{attribute addProperty BoxType "KL6401-0002"}
{attribute addProperty Id "Parameter_StatusAT %I*UINT000Parameter_Input_Data_1AT %I*UDINT000Parameter_Input_Data_2AT %I*UDINT000Parameter_Input_Data_3AT %I*UDINT000Parameter_Input_Data_4AT %I*UDINT000Parameter_Input_Data_5AT %I*UDINT000Parameter_Input_Data_6AT %I*UDINT000Parameter_Input_Data_7AT %I*UDINT000Parameter_Input_Data_8AT %I*UDINT000Parameter_TypeAT %I*USINT000LON_StatusAT %I*USINT000Parameter_ControlAT %Q*UINT000Parameter_Output_Data_1AT %Q*UDINT000Parameter_Output_Data_2AT %Q*UDINT000Parameter_Output_Data_3AT %Q*UDINT000Parameter_Output_Data_4AT %Q*UDINT000Parameter_Output_Data_5AT %Q*UDINT000Parameter_Output_Data_6AT %Q*UDINT000Parameter_Output_Data_7AT %Q*UDINT000Parameter_Output_Data_8AT %Q*UDINT000CMDAT %Q*USINT000IdxAT %Q*USINT000"}
{attribute addProperty CRC "388522448"}
{attribute addProperty SizeInBites "0"}
{attribute addProperty SizeInBytes "0"}
TYPE Channel_172861D0 :
STRUCT
	{attribute addProperty Name "Parameter_Status"}
	Parameter_Status AT %I* : UINT;
	{attribute addProperty Name "Parameter_Input_Data_1"}
	Parameter_Input_Data_1 AT %I* : UDINT;
	{attribute addProperty Name "Parameter_Input_Data_2"}
	Parameter_Input_Data_2 AT %I* : UDINT;
	{attribute addProperty Name "Parameter_Input_Data_3"}
	Parameter_Input_Data_3 AT %I* : UDINT;
	{attribute addProperty Name "Parameter_Input_Data_4"}
	Parameter_Input_Data_4 AT %I* : UDINT;
	{attribute addProperty Name "Parameter_Input_Data_5"}
	Parameter_Input_Data_5 AT %I* : UDINT;
	{attribute addProperty Name "Parameter_Input_Data_6"}
	Parameter_Input_Data_6 AT %I* : UDINT;
	{attribute addProperty Name "Parameter_Input_Data_7"}
	Parameter_Input_Data_7 AT %I* : UDINT;
	{attribute addProperty Name "Parameter_Input_Data_8"}
	Parameter_Input_Data_8 AT %I* : UDINT;
	{attribute addProperty Name "Parameter_Type"}
	Parameter_Type AT %I* : USINT;
	{attribute addProperty Name "LON_Status"}
	LON_Status AT %I* : USINT;
	{attribute addProperty Name "Parameter_Control"}
	Parameter_Control AT %Q* : UINT;
	{attribute addProperty Name "Parameter_Output_Data_1"}
	Parameter_Output_Data_1 AT %Q* : UDINT;
	{attribute addProperty Name "Parameter_Output_Data_2"}
	Parameter_Output_Data_2 AT %Q* : UDINT;
	{attribute addProperty Name "Parameter_Output_Data_3"}
	Parameter_Output_Data_3 AT %Q* : UDINT;
	{attribute addProperty Name "Parameter_Output_Data_4"}
	Parameter_Output_Data_4 AT %Q* : UDINT;
	{attribute addProperty Name "Parameter_Output_Data_5"}
	Parameter_Output_Data_5 AT %Q* : UDINT;
	{attribute addProperty Name "Parameter_Output_Data_6"}
	Parameter_Output_Data_6 AT %Q* : UDINT;
	{attribute addProperty Name "Parameter_Output_Data_7"}
	Parameter_Output_Data_7 AT %Q* : UDINT;
	{attribute addProperty Name "Parameter_Output_Data_8"}
	Parameter_Output_Data_8 AT %Q* : UDINT;
	{attribute addProperty Name "CMD"}
	CMD AT %Q* : USINT;
	{attribute addProperty Name "Idx"}
	Idx AT %Q* : USINT;
END_STRUCT
END_TYPE

(* stored: Version 1.2.0.0, ProductVersion 3.1.4024.9
   DUT Channel_172861D0: Id {05c68a62-4826-4af5-a115-f40f75c8e391} *)
